Yaskawa INFORM job: MCRFEND.JBI

/JOB
//NAME MCRFEND
//POS
///NPOS 0,0,0,0,0,0
//INST
///DATE 2010/10/22 11:00
///ATTR SC,RW,MC
///GROUP1 RB1
NOP
SKILLSND "forcepathend"
END
